FUNCTION_BLOCK FB_AteqResultHandler
VAR_INPUT
	bAutoSeqDone		: BOOL;
	anExchangeZone		: ARRAY[0..127] OF BYTE; // Raw 40-byte ATEQ Last Result block
END_VAR
VAR_IN_OUT	
END_VAR
VAR_OUTPUT
	bLastResultsStored	: BOOL;
	//bFIFOResultsStored	: BOOL;
	stLastResults		: ST_AteqResultsDecoded;
	astLastResults		: ARRAY[0..GVL_AteqConfig.nMaxResultStore] OF ST_AteqResultsDecoded;
END_VAR
VAR
	nOffset 	: INT := 0;
	nTestIndex 	: INT := 0;
END_VAR

IF bAutoSeqDone THEN
    
	// Read and Parse ExchangeZone
    FOR nOffset := 0 TO 127 DO
        M_GetWord(nIndex := nOffset);
        M_GetDWord(nIndex := nOffset);
        M_GetReal(nIndex := nOffset);
    END_FOR

	 M_DecodeLastResults();
	 
    // Store the result once per test
    IF NOT bLastResultsStored AND nTestIndex < GVL_AteqConfig.nMaxResultStore THEN
        astLastResults[nTestIndex] := stLastResults;
        bLastResultsStored := TRUE;
		bAutoSeqDone := FALSE;		
        nTestIndex := nTestIndex + 1; 
    END_IF

ELSE
    bLastResultsStored := FALSE;
END_IF

METHOD M_DecodeLastResults
VAR
	dtTemp 	: DT;
	nOffset : INT;
	wRelayImage : WORD;
END_VAR

// === Word fields ===
stLastResults.nProgramNumber := M_GetWord(0);
stLastResults.nTestType      := M_GetWord(2);
wRelayImage := M_GetWord(4);
stLastResults.nRelayImage := wRelayImage;

// === Relay bits ===
stLastResults.bPassPart          := (wRelayImage AND 16#0001) <> 0;
stLastResults.bFailMaxFlowReject := (wRelayImage AND 16#0002) <> 0;
stLastResults.bFailMinFlowReject := (wRelayImage AND 16#0004) <> 0;
stLastResults.bAlarm             := (wRelayImage AND 16#0008) <> 0;
// Others are reserved

// === Alarm code ===
stLastResults.nAlarmCode := M_GetWord(6);

// === Real + DWORD Unit code pairs ===
stLastResults.fPressure              := M_GetReal(8) / 1000.0;
stLastResults.nPressureUnitCode      := M_GetDWord(12) / 1000;

stLastResults.fLeak                  := M_GetReal(16) / 10000.0;
stLastResults.nLeakUnitCode          := M_GetDWord(20) / 1000;

stLastResults.fPressurePiezo2        := M_GetReal(24) / 1000.0;
stLastResults.nPressurePiezo2UnitCode:= M_GetDWord(28) / 1000;

stLastResults.fTestCheckResult       := M_GetReal(32) / 1000.0;
stLastResults.nTestCheckResultUnitCode := M_GetDWord(36) / 1000;

stLastResults.fLargeLeak             := M_GetReal(40) / 1000.0;
stLastResults.nLargeLeakUnitCode     := M_GetDWord(44) / 1000;

stLastResults.fPaLeakResult          := M_GetReal(48) / 1000.0;

// === Reserved WORDs (10 WORDs from byte 52 to 71) ===
FOR nOffset := 0 TO 9 DO
	stLastResults.aReserved[27 + nOffset] := M_GetWord(52 + nOffset * 2);
END_FOR

// === Environmental ===
stLastResults.fAtmPressure  := M_GetReal(72) / 1000.0;
stLastResults.fTempCelcius  := M_GetReal(76) / 1000.0;

// === Timestamp (DT) ===
stLastResults.dtTestTimeStamp := GVL_Controller.dtSystemTime;
END_METHOD

METHOD PRIVATE M_GetDWord : DWORD
VAR_INPUT
	nIndex : INT;
END_VAR
VAR
	nLowWord  : WORD;
	nHighWord : WORD;
END_VAR

nLowWord := M_GetWord(nIndex := nIndex);
nHighWord := M_GetWord(nIndex := nIndex + 2);
IF GVL_AteqConfig.eDeviceEndianSetTo = E_AteqEndianType.LittleEndian THEN
	M_GetDword := SHL(WORD_TO_DWORD(nLowWord), 16) OR WORD_TO_DWORD(nHighWord);
ELSE
	M_GetDword := SHL(WORD_TO_DWORD(nHighWord), 16) OR WORD_TO_DWORD(nLowWord);
END_IF
END_METHOD

METHOD PRIVATE M_GetReal : REAL
VAR_INPUT
	nIndex : INT;	
END_VAR
VAR
	nDWord : DWORD;
END_VAR
nDWord := M_GetDWord(nIndex := nIndex);
M_GetReal := DWORD_TO_REAL(nDWord);
END_METHOD

METHOD PRIVATE M_GetWord : WORD
VAR_INPUT
	nIndex : INT;
END_VAR

IF GVL_AteqConfig.eDeviceEndianSetTo = E_AteqEndianType.LittleEndian THEN
	M_GetWord := SHL(BYTE_TO_WORD(anExchangeZone[nIndex]), 8) OR BYTE_TO_WORD(anExchangeZone[nIndex + 1]);
ELSE
	M_GetWord := BYTE_TO_WORD(anExchangeZone[nIndex]) OR SHL(BYTE_TO_WORD(anExchangeZone[nIndex + 1]), 8);
END_IF
END_METHOD

END_FUNCTION_BLOCK

(* stored: Version 1.1.0.1
   POU FB_AteqResultHandler: Id {83a39566-cc01-4a56-a640-0780618ac137}, SpecialFunc None
   Method M_DecodeLastResults: Id {ae5e062d-88f2-44cf-8bfc-3c173c4914c7}
   Method M_GetDWord: Id {ae3ff039-bb3d-4e21-88fd-0677b0274f55}
   Method M_GetReal: Id {7f230d3b-3725-4a01-ae93-b74613e3223d}
   Method M_GetWord: Id {1767a00b-de76-4571-b2d0-10fc51192ebe} *)
